// TIA Portal V18 export
FUNCTION "Boiler_Main" : Void   // FC1010, LAD
{ S7_Optimized_Access := 'TRUE' }
VERSION : 0.1
// stored: AutoNumber false, IsIECCheckEnabled false, SetENOAutomatically false, UDAEnableTagReadback false
BEGIN

REGION Network 1
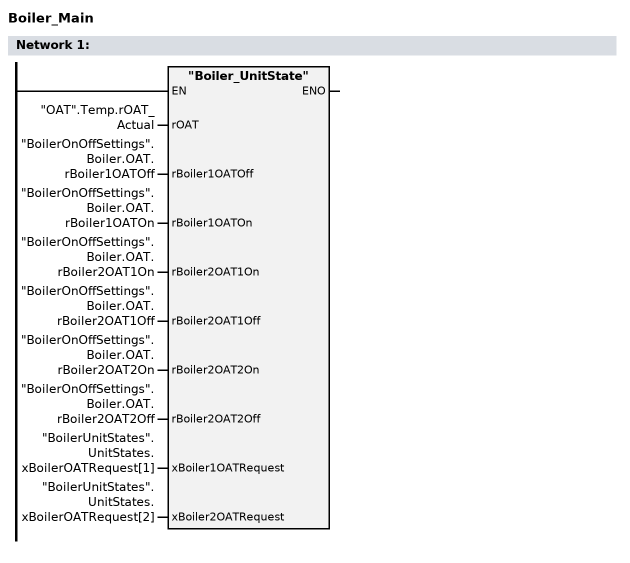
   RUNG wire#powerrail
      "Boiler_UnitState"(rOAT := "OAT".Temp.rOAT_Actual, rBoiler1OATOff := "BoilerOnOffSettings".Boiler.OAT.rBoiler1OATOff, rBoiler1OATOn := "BoilerOnOffSettings".Boiler.OAT.rBoiler1OATOn, rBoiler2OAT1On := "BoilerOnOffSettings".Boiler.OAT.rBoiler2OAT1On, rBoiler2OAT1Off := "BoilerOnOffSettings".Boiler.OAT.rBoiler2OAT1Off, rBoiler2OAT2On := "BoilerOnOffSettings".Boiler.OAT.rBoiler2OAT2On, rBoiler2OAT2Off := "BoilerOnOffSettings".Boiler.OAT.rBoiler2OAT2Off, xBoiler1OATRequest := "BoilerUnitStates".UnitStates.xBoilerOATRequest[1], xBoiler2OATRequest := "BoilerUnitStates".UnitStates.xBoilerOATRequest[2])
   END_RUNG
   // the same network as SCL:
   "Boiler_UnitState"(rOAT := "OAT".Temp.rOAT_Actual,
                      rBoiler1OATOff := "BoilerOnOffSettings".Boiler.OAT.rBoiler1OATOff,
                      rBoiler1OATOn := "BoilerOnOffSettings".Boiler.OAT.rBoiler1OATOn,
                      rBoiler2OAT1On := "BoilerOnOffSettings".Boiler.OAT.rBoiler2OAT1On,
                      rBoiler2OAT1Off := "BoilerOnOffSettings".Boiler.OAT.rBoiler2OAT1Off,
                      rBoiler2OAT2On := "BoilerOnOffSettings".Boiler.OAT.rBoiler2OAT2On,
                      rBoiler2OAT2Off := "BoilerOnOffSettings".Boiler.OAT.rBoiler2OAT2Off,
                      xBoiler1OATRequest := "BoilerUnitStates".UnitStates.xBoilerOATRequest[1],
                      xBoiler2OATRequest := "BoilerUnitStates".UnitStates.xBoilerOATRequest[2]);
END_REGION
END_FUNCTION
